{attribute 'qualified_only'}
VAR_GLOBAL
	Analog_Outputs_Curr AT %Q* : ARRAY[1..2] OF INT;
	Analog_Outputs_Curr_Values : ARRAY[1..2] OF REAL;
END_VAR

(* stored: Version 1.1.0.1, ProductVersion 3.1.4024.12
   GVL GVL: Id {d23ebe54-3032-44e2-a33a-beac0c680307} *)
